// TIA Portal V18 export
DATA_BLOCK "PAutoPrePos"   // DB40
{ S7_Optimized_Access := 'TRUE' }
VERSION : 0.1
// stored: AutoNumber true, IsOnlyStoredInLoadMemory false, IsRetainMemResEnabled false, IsWriteProtectedInAS false, MemoryReserve 100
   VAR RETAIN
      "Boing 737_PBB" : Array[0..1] of Real;
      "Boing 737-Max_PBB" : Array[0..1] of Real;
      "MD 80 & 90 Series" : Array[0..1] of Real;
      "Airbus A318/319/320" : Array[0..1] of Real;
      Embraer : Array[0..1] of Real;
      "Airbus A300/310/330/340" : Array[0..1] of Real;
      "Airbus A350" : Array[0..1] of Real;
      "Boing 747/777" : Array[0..1] of Real;
   END_VAR
BEGIN
   "Boing 737_PBB"[0] := 2.77;
   "Boing 737_PBB"[1] := 40.0;
   "Boing 737-Max_PBB"[0] := 3.07;
   "Boing 737-Max_PBB"[1] := 22.0;
   "MD 80 & 90 Series"[0] := 2.4;
   "MD 80 & 90 Series"[1] := 30.0;
   "Airbus A318/319/320"[0] := 3.48;
   "Airbus A318/319/320"[1] := 48.0;
   Embraer[0] := 2.75;
   Embraer[1] := 51.0;
   "Airbus A300/310/330/340"[0] := 4.76;
   "Airbus A300/310/330/340"[1] := 35.0;
   "Airbus A350"[0] := 5.0;
   "Airbus A350"[1] := 22.0;
   "Boing 747/777"[0] := 5.0;
   "Boing 747/777"[1] := 26.0;
END_DATA_BLOCK
